RoboDK station: Sheet A.rdk

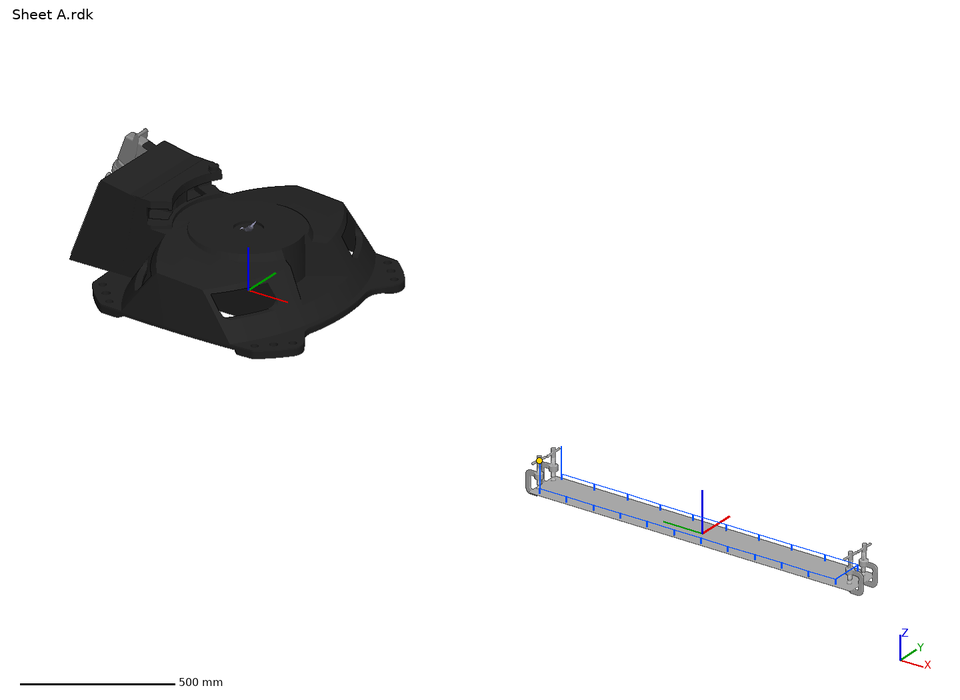
[picture v0: the station drawn from its stored meshes, robots at their saved joint values, targets as dots, program paths as lines]
Station Sheet A (saved by RoboDK 5.2.3). Poses are relative to the parent item; angles as X-Y-Z fixed-axis rotations.
  - frame KUKA KR 210 R2700 extra Base at (0, 0, 0) mm
    - robot KUKA KR 210 R2700 extra: 6 axes, payload 210 kg, reach 2696 mm, repeatability 0.06 mm, weight 1068 kg
        joint limits [-185, -140, -120, -350, -125, -350] to [185, -5, 155, 350, 125, 350]; home [0, -90, 90, 0, 0, 0]; saved at [-3.864, -30.644, 139.201, -182.881, 57.526, -181.457]
      - tool Spindle, TCP at (32, 0, 260) mm, rotated rx 0 ry 39 rz 0 deg, size 157.3 x 72 x 259.9 mm
  - frame Frame 2 at (1788.65, 0, -372.68) mm, rotated rx 0 ry 0 rz 90 deg
    - object Box 2 - Sheet A at (0, 0, 0) mm, size 148.8 x 1269.1 x 0.8 mm, geometry from Box 2 - Sheet A.stl
    - object sheetAbox2 at (0, 0, 0) mm, 22 curves, geometry from Point 22
  - machining project Point settings: C:/Users/jbert/AppData/Local/Temp/Box 2 - Sheet A.stl | rotZ(0) | rotX(0)*rotY(0) | rotz(0) | onStart | onPathStart | onApproach | onPoint | onRetract | onFinish | SetRPM(%1) | SetTool(%1) | Extruder(%1) | default | default | OutOnMov(%1) | OutOffMov(%1) | onPathFinish | M_RunCode(%1)
  - program Point (121 instructions, listed below)
  - object FinalClamp at (1174.79, 36.64, -311.7) mm, rotated rx 86.88 ry 89.77 rz 180 deg, size 145.3 x 71.1 x 72 mm, geometry from FinalClamp.stp
  - object FinalClamp2 at (1170.74, -38.12, -311.48) mm, rotated rx -137.35 ry 88.73 rz -50.56 deg, size 145.3 x 71.1 x 72 mm, geometry from FinalClamp.stp
  - object FinalClamp3 at (2397.74, -40.83, -309.24) mm, rotated rx -89.23 ry 87.74 rz 180 deg, size 145.3 x 71.1 x 72 mm, geometry from FinalClamp.stp
  - object FinalClamp4 at (2398.73, 35.43, -310.05) mm, rotated rx -99.75 ry 86.92 rz 171.37 deg, size 145.3 x 71.1 x 72 mm, geometry from FinalClamp.stp
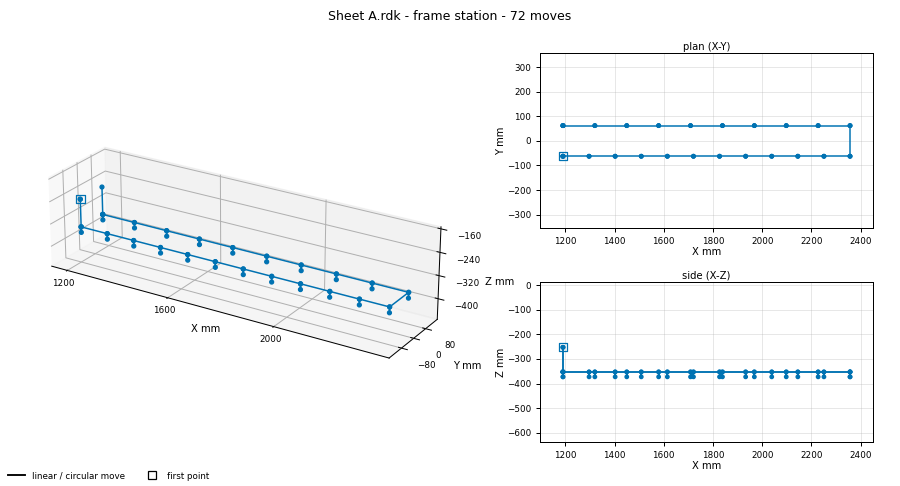
[picture p0: tool path of Sheet A.rdk in frame station, 72 of 72 moves have a stored position in this frame; points joined in program order, loops and branches not executed]

--- program Point (robot KUKA KR 210 R2700 extra) ---
  Smooth(7)
  Set speed (1000.0 mm/s)
  Set Ref.: Frame 2
  Set Tool: Spindle
  Show Spindle
  MoveJ 1 to (-62.4, 598.04, 120) mm, rotated rx 180 ry 0 rz 90 deg; joints [3.895, -30.645, 139.2, -177.096, 57.523, -178.532]
  MoveL 2 to (-62.4, 598.04, 120) mm, rotated rx 180 ry 0 rz 90 deg; joints [3.895, -30.645, 139.2, -177.096, 57.523, -178.532]
  MoveL 3 to (-62.4, 598.04, 20) mm, rotated rx -180 ry 0 rz 90 deg; joints [3.895, -23.568, 135.456, -177.195, 60.853, -178.339]
  MoveL 4 to (-62.4, 598.04, 20) mm, rotated rx -180 ry 0 rz 90 deg; joints [3.895, -23.568, 135.456, -177.195, 60.853, -178.339]
  Set speed (50.0 mm/s)
  MoveL 5 to (-62.4, 598.04, 0) mm, rotated rx -180 ry 0 rz 90 deg; joints [3.895, -22.234, 134.667, -177.209, 61.397, -178.308]
  MoveL 6 to (-62.4, 598.04, 20) mm, rotated rx -180 ry 0 rz 90 deg; joints [3.895, -23.568, 135.456, -177.195, 60.853, -178.339]
  Set speed (1000.0 mm/s)
  MoveL 7 to (-62.4, 492.04, 20) mm, rotated rx 180 ry 0 rz 90 deg; joints [3.492, -26.21, 131.565, -177.296, 54.334, -178.862]
  Set speed (50.0 mm/s)
  MoveL 8 to (-62.4, 492.04, 0) mm, rotated rx 180 ry 0 rz 90 deg; joints [3.492, -24.908, 130.828, -177.314, 54.898, -178.83]
  MoveL 9 to (-62.4, 492.04, 20) mm, rotated rx 180 ry 0 rz 90 deg; joints [3.492, -26.21, 131.565, -177.296, 54.334, -178.862]
  Set speed (1000.0 mm/s)
  MoveL 10 to (-62.4, 386.04, 20) mm, rotated rx -180 ry 0 rz 90 deg; joints [3.165, -27.947, 127.307, -177.335, 48.348, -179.311]
  Set speed (50.0 mm/s)
  MoveL 11 to (-62.4, 386.04, 0) mm, rotated rx 180 ry 0 rz 90 deg; joints [3.165, -26.693, 126.615, -177.358, 48.91, -179.277]
  MoveL 12 to (-62.4, 386.04, 20) mm, rotated rx -180 ry 0 rz 90 deg; joints [3.165, -27.947, 127.307, -177.335, 48.348, -179.311]
  Set speed (1000.0 mm/s)
  MoveL 13 to (-62.4, 280.04, 20) mm, rotated rx 180 ry 0 rz 90 deg; joints [2.894, -28.927, 122.725, -177.32, 42.793, -179.718]
  Set speed (50.0 mm/s)
  MoveL 14 to (-62.4, 280.04, 0) mm, rotated rx -180 ry 0 rz 90 deg; joints [2.894, -27.727, 122.073, -177.347, 43.341, -179.681]
  MoveL 15 to (-62.4, 280.04, 20) mm, rotated rx 180 ry 0 rz 90 deg; joints [2.894, -28.927, 122.725, -177.32, 42.793, -179.718]
  Set speed (1000.0 mm/s)
  MoveL 16 to (-62.4, 174.04, 20) mm, rotated rx -180 ry 0 rz 90 deg; joints [2.665, -29.269, 117.846, -177.25, 37.578, -180.109]
  Set speed (50.0 mm/s)
  MoveL 17 to (-62.4, 174.04, 0) mm, rotated rx -180 ry 0 rz 90 deg; joints [2.665, -28.124, 117.228, -177.282, 38.104, -180.068]
  MoveL 18 to (-62.4, 174.04, 20) mm, rotated rx -180 ry 0 rz 90 deg; joints [2.665, -29.269, 117.846, -177.25, 37.578, -180.109]
  Set speed (1000.0 mm/s)
  MoveL 19 to (-62.4, 68.04, 20) mm, rotated rx -180 ry 0 rz 90 deg; joints [2.47, -29.067, 112.681, -177.116, 32.62, -180.51]
  Set speed (50.0 mm/s)
  MoveL 20 to (-62.4, 68.04, 0) mm, rotated rx 180 ry 0 rz 90 deg; joints [2.47, -27.977, 112.09, -177.155, 33.12, -180.463]
  MoveL 21 to (-62.4, 68.04, 20) mm, rotated rx -180 ry 0 rz 90 deg; joints [2.47, -29.067, 112.681, -177.116, 32.62, -180.51]
  Set speed (1000.0 mm/s)
  MoveL 22 to (-62.4, -37.96, 20) mm, rotated rx -180 ry 0 rz 90 deg; joints [2.302, -28.392, 107.227, -176.899, 27.847, -180.954]
  Set speed (50.0 mm/s)
  MoveL 23 to (-62.4, -37.96, 0) mm, rotated rx -180 ry 0 rz 90 deg; joints [2.302, -27.352, 106.659, -176.946, 28.318, -180.9]
  MoveL 24 to (-62.4, -37.96, 20) mm, rotated rx -180 ry 0 rz 90 deg; joints [2.302, -28.392, 107.227, -176.899, 27.847, -180.954]
  Set speed (1000.0 mm/s)
  MoveL 25 to (-62.4, -143.96, 20) mm, rotated rx 180 ry 0 rz 90 deg; joints [2.155, -27.292, 101.47, -176.556, 23.195, -181.491]
  Set speed (50.0 mm/s)
  MoveL 26 to (-62.4, -143.96, 0) mm, rotated rx -180 ry 0 rz 90 deg; joints [2.155, -26.298, 100.917, -176.617, 23.636, -181.425]
  MoveL 27 to (-62.4, -143.96, 20) mm, rotated rx 180 ry 0 rz 90 deg; joints [2.155, -27.292, 101.47, -176.556, 23.195, -181.491]
  Set speed (1000.0 mm/s)
  MoveL 28 to (-62.4, -249.96, 20) mm, rotated rx 180 ry 0 rz 90 deg; joints [2.025, -25.799, 95.378, -176.002, 18.604, -182.215]
  Set speed (50.0 mm/s)
  MoveL 29 to (-62.4, -249.96, 0) mm, rotated rx -180 ry 0 rz 90 deg; joints [2.025, -24.845, 94.835, -176.086, 19.014, -182.127]
  MoveL 30 to (-62.4, -249.96, 20) mm, rotated rx 180 ry 0 rz 90 deg; joints [2.025, -25.799, 95.378, -176.002, 18.604, -182.215]
  Set speed (1000.0 mm/s)
  MoveL 31 to (-62.4, -355.96, 20) mm, rotated rx 180 ry 0 rz 90 deg; joints [1.911, -23.923, 88.902, -175.029, 14.014, -183.338]
  Set speed (50.0 mm/s)
  MoveL 32 to (-62.4, -355.96, 0) mm, rotated rx -180 ry 0 rz 90 deg; joints [1.911, -23.004, 88.364, -175.158, 14.393, -183.206]
  MoveL 33 to (-62.4, -355.96, 20) mm, rotated rx 180 ry 0 rz 90 deg; joints [1.911, -23.923, 88.902, -175.029, 14.014, -183.338]
  Set speed (1000.0 mm/s)
  MoveL 34 to (-62.4, -461.96, 20) mm, rotated rx -180 ry 0 rz 90 deg; joints [1.808, -21.656, 81.968, -172.992, 9.367, -185.51]
  Set speed (50.0 mm/s)
  MoveL 35 to (-62.4, -461.96, 0) mm, rotated rx -180 ry 0 rz 90 deg; joints [1.808, -20.767, 81.427, -173.24, 9.712, -185.259]
  MoveL 36 to (-62.4, -461.96, 20) mm, rotated rx -180 ry 0 rz 90 deg; joints [1.808, -21.656, 81.968, -172.992, 9.367, -185.51]
  Set speed (1000.0 mm/s)
  MoveL 37 to (-62.4, -567.96, 20) mm, rotated rx 180 ry 0 rz 90 deg; joints [1.716, -18.966, 74.465, -166.45, 4.614, -192.174]
  Set speed (50.0 mm/s)
  MoveL 38 to (-62.4, -567.96, 0) mm, rotated rx -180 ry 0 rz 90 deg; joints [1.716, -18.1, 73.911, -167.301, 4.918, -191.32]
  MoveL 39 to (-62.4, -567.96, 20) mm, rotated rx 180 ry 0 rz 90 deg; joints [1.716, -18.966, 74.465, -166.45, 4.614, -192.174]
  Set speed (1000.0 mm/s)
  MoveL 40 to (61.9, -567.96, 20) mm, rotated rx -180 ry 0 rz 90 deg; joints [-1.703, -18.967, 74.466, -193.443, 4.613, -167.922]
  Set speed (50.0 mm/s)
  MoveL 41 to (61.9, -567.96, 0) mm, rotated rx -180 ry 0 rz 90 deg; joints [-1.703, -18.1, 73.912, -192.599, 4.917, -168.77]
  MoveL 42 to (61.9, -567.96, 20) mm, rotated rx -180 ry 0 rz 90 deg; joints [-1.703, -18.967, 74.466, -193.443, 4.613, -167.922]
  Set speed (1000.0 mm/s)
  MoveL 43 to (61.9, -438.4, 20) mm, rotated rx -180 ry 0 rz 90 deg; joints [-1.815, -22.195, 83.555, -186.336, 10.408, -175.179]
  Set speed (50.0 mm/s)
  MoveL 44 to (61.9, -438.4, 0) mm, rotated rx 180 ry 0 rz 90 deg; joints [-1.815, -21.3, 83.015, -186.13, 10.761, -175.388]
  MoveL 45 to (61.9, -438.4, 20) mm, rotated rx -180 ry 0 rz 90 deg; joints [-1.815, -22.195, 83.555, -186.336, 10.408, -175.179]
  Set speed (1000.0 mm/s)
  MoveL 46 to (61.9, -308.85, 20) mm, rotated rx -180 ry 0 rz 90 deg; joints [-1.944, -24.804, 91.832, -184.427, 16.058, -177.256]
  Set speed (50.0 mm/s)
  MoveL 47 to (61.9, -308.85, 0) mm, rotated rx 180 ry 0 rz 90 deg; joints [-1.944, -23.871, 91.293, -184.324, 16.451, -177.364]
  MoveL 48 to (61.9, -308.85, 20) mm, rotated rx -180 ry 0 rz 90 deg; joints [-1.944, -24.804, 91.832, -184.427, 16.058, -177.256]
  Set speed (1000.0 mm/s)
  MoveL 49 to (61.9, -179.29, 20) mm, rotated rx 180 ry 0 rz 90 deg; joints [-2.093, -26.838, 99.48, -183.57, 21.661, -178.309]
  Set speed (50.0 mm/s)
  MoveL 50 to (61.9, -179.29, 0) mm, rotated rx -180 ry 0 rz 90 deg; joints [-2.093, -25.857, 98.931, -183.503, 22.092, -178.38]
  MoveL 51 to (61.9, -179.29, 20) mm, rotated rx 180 ry 0 rz 90 deg; joints [-2.093, -26.838, 99.48, -183.57, 21.661, -178.309]
  Set speed (1000.0 mm/s)
  MoveL 52 to (61.9, -49.74, 20) mm, rotated rx 180 ry 0 rz 90 deg; joints [-2.266, -28.29, 106.604, -183.107, 27.326, -179]
  Set speed (50.0 mm/s)
  MoveL 53 to (61.9, -49.74, 0) mm, rotated rx 180 ry 0 rz 90 deg; joints [-2.266, -27.255, 106.037, -183.059, 27.794, -179.055]
  MoveL 54 to (61.9, -49.74, 20) mm, rotated rx 180 ry 0 rz 90 deg; joints [-2.266, -28.29, 106.604, -183.107, 27.326, -179]
  Set speed (1000.0 mm/s)
  MoveL 55 to (61.9, 79.82, 20) mm, rotated rx 180 ry 0 rz 90 deg; joints [-2.47, -29.114, 113.27, -182.842, 33.162, -179.54]
  Set speed (50.0 mm/s)
  MoveL 56 to (61.9, 79.82, 0) mm, rotated rx 180 ry 0 rz 90 deg; joints [-2.47, -28.018, 112.676, -182.805, 33.664, -179.585]
  MoveL 57 to (61.9, 79.82, 20) mm, rotated rx 180 ry 0 rz 90 deg; joints [-2.47, -29.114, 113.27, -182.842, 33.162, -179.54]
  Set speed (1000.0 mm/s)
  MoveL 58 to (61.9, 209.38, 20) mm, rotated rx -180 ry 0 rz 90 deg; joints [-2.715, -29.22, 119.506, -182.699, 39.286, -180.021]
  Set speed (50.0 mm/s)
  MoveL 59 to (61.9, 209.38, 0) mm, rotated rx -180 ry 0 rz 90 deg; joints [-2.715, -28.056, 118.877, -182.668, 39.82, -180.061]
  MoveL 60 to (61.9, 209.38, 20) mm, rotated rx -180 ry 0 rz 90 deg; joints [-2.715, -29.22, 119.506, -182.699, 39.286, -180.021]
  Set speed (1000.0 mm/s)
  MoveL 61 to (61.9, 338.93, 20) mm, rotated rx 180 ry 0 rz 90 deg; joints [-3.014, -28.468, 125.31, -182.644, 45.833, -180.5]
  Set speed (50.0 mm/s)
  MoveL 62 to (61.9, 338.93, 0) mm, rotated rx 180 ry 0 rz 90 deg; joints [-3.014, -27.237, 124.637, -182.619, 46.39, -180.536]
  MoveL 63 to (61.9, 338.93, 20) mm, rotated rx 180 ry 0 rz 90 deg; joints [-3.014, -28.468, 125.31, -182.644, 45.833, -180.5]
  Set speed (1000.0 mm/s)
  MoveL 64 to (61.9, 468.49, 20) mm, rotated rx 180 ry 0 rz 90 deg; joints [-3.386, -26.668, 130.65, -182.669, 52.964, -181.024]
  Set speed (50.0 mm/s)
  MoveL 65 to (61.9, 468.49, 0) mm, rotated rx 180 ry 0 rz 90 deg; joints [-3.386, -25.375, 129.923, -182.65, 53.528, -181.057]
  MoveL 66 to (61.9, 468.49, 20) mm, rotated rx 180 ry 0 rz 90 deg; joints [-3.386, -26.668, 130.65, -182.669, 52.964, -181.024]
  Set speed (1000.0 mm/s)
  MoveL 67 to (61.9, 598.04, 20) mm, rotated rx 180 ry 0 rz 90 deg; joints [-3.864, -23.567, 135.457, -182.783, 60.855, -181.648]
  Set speed (50.0 mm/s)
  MoveL 68 to (61.9, 598.04, 0) mm, rotated rx -180 ry 0 rz 90 deg; joints [-3.864, -22.233, 134.668, -182.768, 61.4, -181.678]
  MoveL 69 to (61.9, 598.04, 20) mm, rotated rx 180 ry 0 rz 90 deg; joints [-3.864, -23.567, 135.457, -182.783, 60.855, -181.648]
  MoveL 70 to (61.9, 598.04, 20) mm, rotated rx 180 ry 0 rz 90 deg; joints [-3.864, -23.567, 135.457, -182.783, 60.855, -181.648]
  Set speed (1000.0 mm/s)
  MoveL 71 to (61.9, 598.04, 20) mm, rotated rx 180 ry 0 rz 90 deg; joints [-3.864, -23.567, 135.457, -182.783, 60.855, -181.648]
  MoveL 72 to (61.9, 598.04, 120) mm, rotated rx 180 ry 0 rz 90 deg; joints [-3.864, -30.644, 139.201, -182.881, 57.526, -181.457]
